FUNCTION_BLOCK FB_Blinker
VAR_INPUT
	Period	: TIME;
END_VAR
VAR_OUTPUT
	Output	: BOOL;
	fET		: LREAL;
END_VAR
VAR
	Timer1: TON;
END_VAR

Timer1(In := NOT Timer1.Q, PT := Period);
Output	:= Period/2 > Timer1.ET;
fET		:= TIME_TO_LREAL(Timer1.ET);

END_FUNCTION_BLOCK

(* stored: Version 1.1.0.1, ProductVersion 3.1.4024.4
   POU FB_Blinker: Id {092761fc-1b18-48a1-9383-71c4cc0886e6}, SpecialFunc None *)
